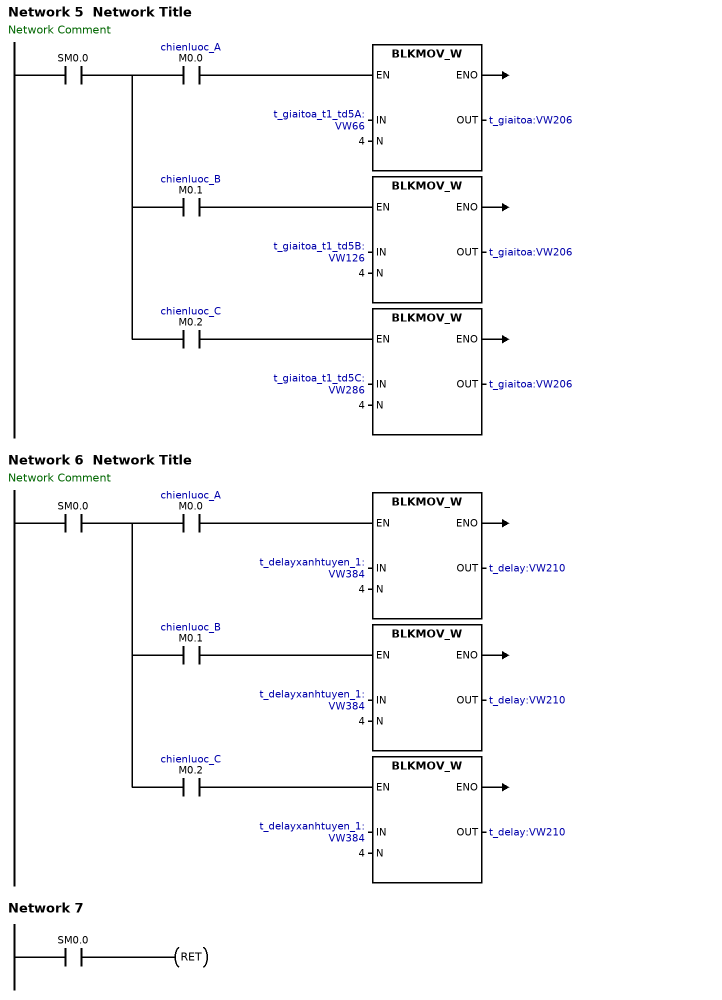
[picture p24: SBR7 networks 5-7]
Network 5 // Network Title
// Network Comment
LD     SM0.0
LPS
A      chienluoc_A:M0.0
BMW    t_giaitoa_t1_td5A:VW66, t_giaitoa:VW206, 4
LRD
A      chienluoc_B:M0.1
BMW    t_giaitoa_t1_td5B:VW126, t_giaitoa:VW206, 4
LPP
A      chienluoc_C:M0.2
BMW    t_giaitoa_t1_td5C:VW286, t_giaitoa:VW206, 4
Network 6 // Network Title
// Network Comment
LD     SM0.0
LPS
A      chienluoc_A:M0.0
BMW    t_delayxanhtuyen_1:VW384, t_delay:VW210, 4
LRD
A      chienluoc_B:M0.1
BMW    t_delayxanhtuyen_1:VW384, t_delay:VW210, 4
LPP
A      chienluoc_C:M0.2
BMW    t_delayxanhtuyen_1:VW384, t_delay:VW210, 4
Network 7
LD     SM0.0
CRET
END_SUBROUTINE_BLOCK

SUBROUTINE_BLOCK thoidiem6:SBR8
TITLE=SUBROUTINE COMMENTS
BEGIN
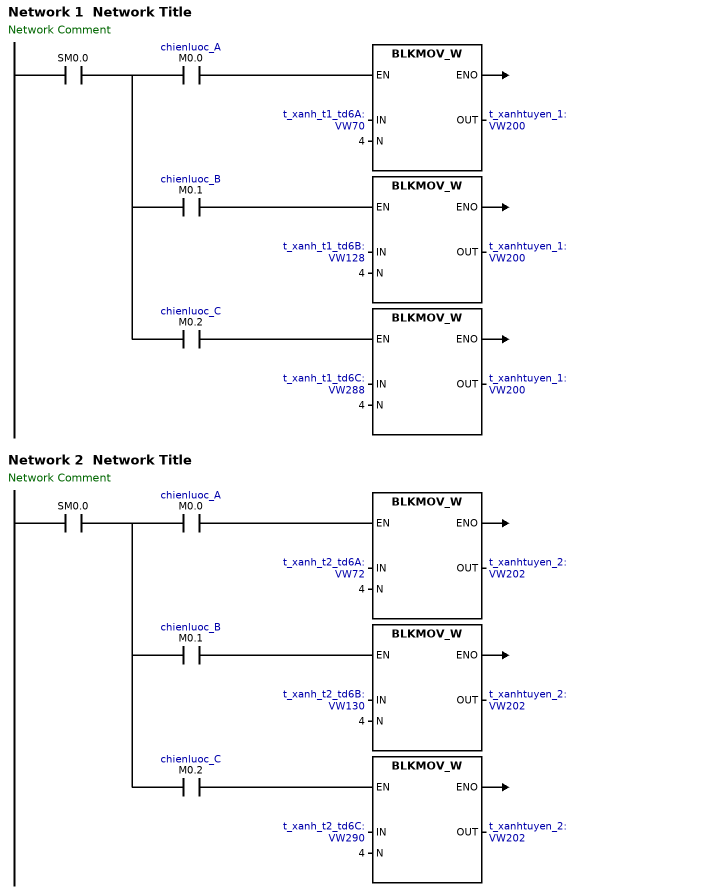
Network 1 // Network Title
// Network Comment
LD     SM0.0
LPS
A      chienluoc_A:M0.0
BMW    t_xanh_t1_td6A:VW70, t_xanhtuyen_1:VW200, 4
LRD
A      chienluoc_B:M0.1
BMW    t_xanh_t1_td6B:VW128, t_xanhtuyen_1:VW200, 4
LPP
A      chienluoc_C:M0.2
BMW    t_xanh_t1_td6C:VW288, t_xanhtuyen_1:VW200, 4
Network 2 // Network Title
// Network Comment
LD     SM0.0
LPS
A      chienluoc_A:M0.0
BMW    t_xanh_t2_td6A:VW72, t_xanhtuyen_2:VW202, 4
LRD
A      chienluoc_B:M0.1
BMW    t_xanh_t2_td6B:VW130, t_xanhtuyen_2:VW202, 4
LPP
A      chienluoc_C:M0.2
BMW    t_xanh_t2_td6C:VW290, t_xanhtuyen_2:VW202, 4
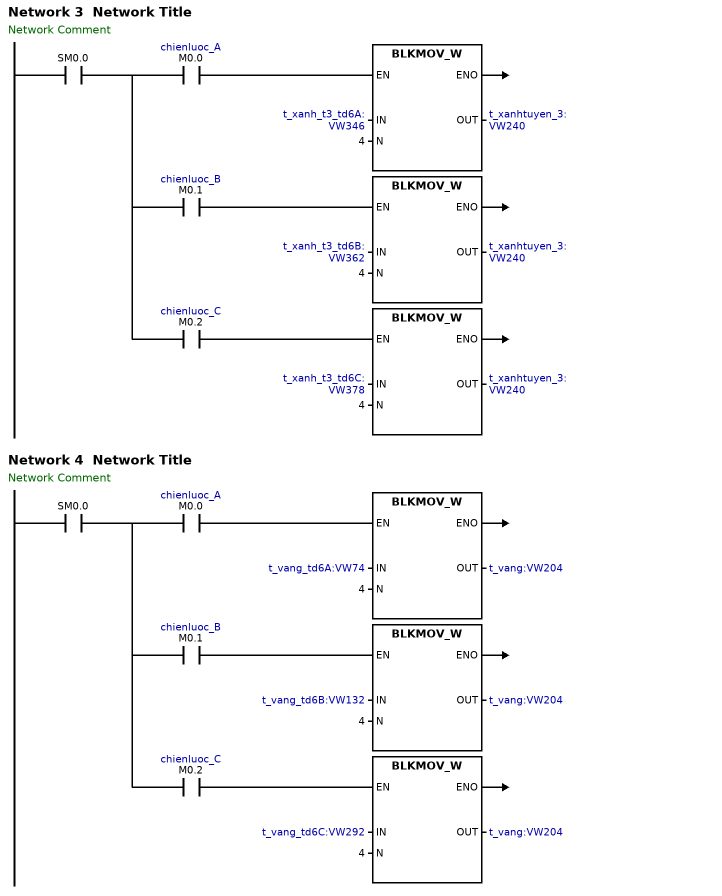
Network 3 // Network Title
// Network Comment
LD     SM0.0
LPS
A      chienluoc_A:M0.0
BMW    t_xanh_t3_td6A:VW346, t_xanhtuyen_3:VW240, 4
LRD
A      chienluoc_B:M0.1
BMW    t_xanh_t3_td6B:VW362, t_xanhtuyen_3:VW240, 4
LPP
A      chienluoc_C:M0.2
BMW    t_xanh_t3_td6C:VW378, t_xanhtuyen_3:VW240, 4
Network 4 // Network Title
// Network Comment
LD     SM0.0
LPS
A      chienluoc_A:M0.0
BMW    t_vang_td6A:VW74, t_vang:VW204, 4
LRD
A      chienluoc_B:M0.1
BMW    t_vang_td6B:VW132, t_vang:VW204, 4
LPP
A      chienluoc_C:M0.2
BMW    t_vang_td6C:VW292, t_vang:VW204, 4
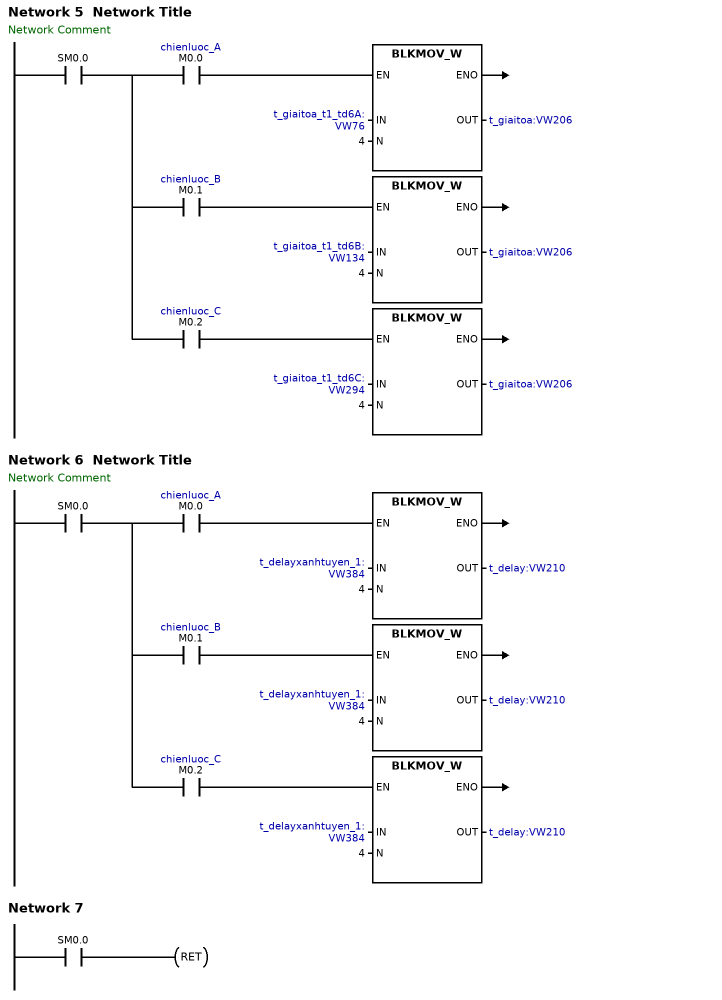
Network 5 // Network Title
// Network Comment
LD     SM0.0
LPS
A      chienluoc_A:M0.0
BMW    t_giaitoa_t1_td6A:VW76, t_giaitoa:VW206, 4
LRD
A      chienluoc_B:M0.1
BMW    t_giaitoa_t1_td6B:VW134, t_giaitoa:VW206, 4
LPP
A      chienluoc_C:M0.2
BMW    t_giaitoa_t1_td6C:VW294, t_giaitoa:VW206, 4
Network 6 // Network Title
// Network Comment
LD     SM0.0
LPS
A      chienluoc_A:M0.0
BMW    t_delayxanhtuyen_1:VW384, t_delay:VW210, 4
LRD
A      chienluoc_B:M0.1
BMW    t_delayxanhtuyen_1:VW384, t_delay:VW210, 4
LPP
A      chienluoc_C:M0.2
BMW    t_delayxanhtuyen_1:VW384, t_delay:VW210, 4
Network 7
LD     SM0.0
CRET
END_SUBROUTINE_BLOCK

SUBROUTINE_BLOCK thoidiem7:SBR9
TITLE=SUBROUTINE COMMENTS
BEGIN
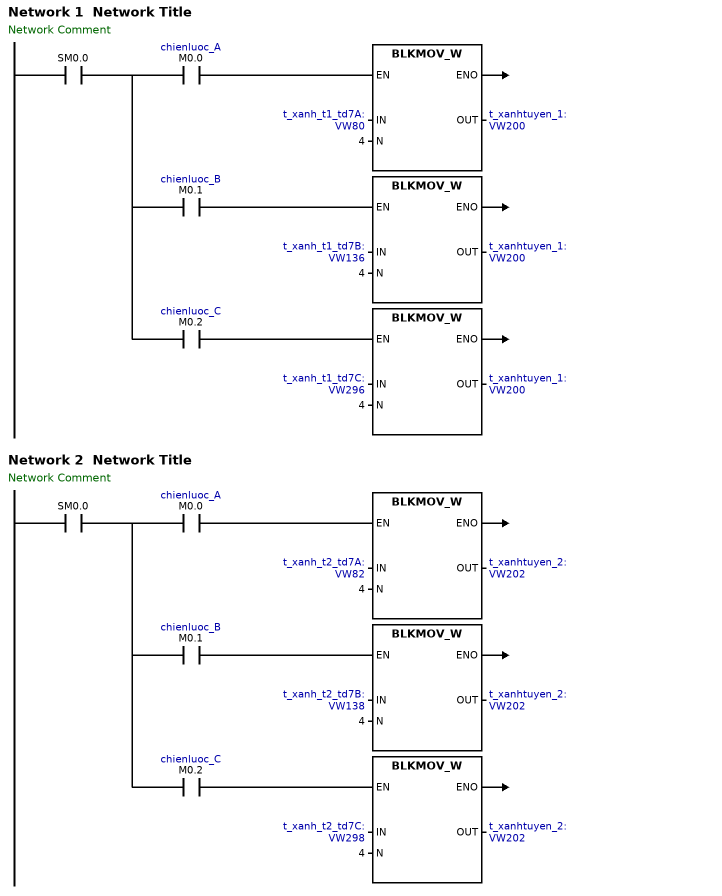
Network 1 // Network Title
// Network Comment
LD     SM0.0
LPS
A      chienluoc_A:M0.0
BMW    t_xanh_t1_td7A:VW80, t_xanhtuyen_1:VW200, 4
LRD
A      chienluoc_B:M0.1
BMW    t_xanh_t1_td7B:VW136, t_xanhtuyen_1:VW200, 4
LPP
A      chienluoc_C:M0.2
BMW    t_xanh_t1_td7C:VW296, t_xanhtuyen_1:VW200, 4
Network 2 // Network Title
// Network Comment
LD     SM0.0
LPS
A      chienluoc_A:M0.0
BMW    t_xanh_t2_td7A:VW82, t_xanhtuyen_2:VW202, 4
LRD
A      chienluoc_B:M0.1
BMW    t_xanh_t2_td7B:VW138, t_xanhtuyen_2:VW202, 4
LPP
A      chienluoc_C:M0.2
BMW    t_xanh_t2_td7C:VW298, t_xanhtuyen_2:VW202, 4
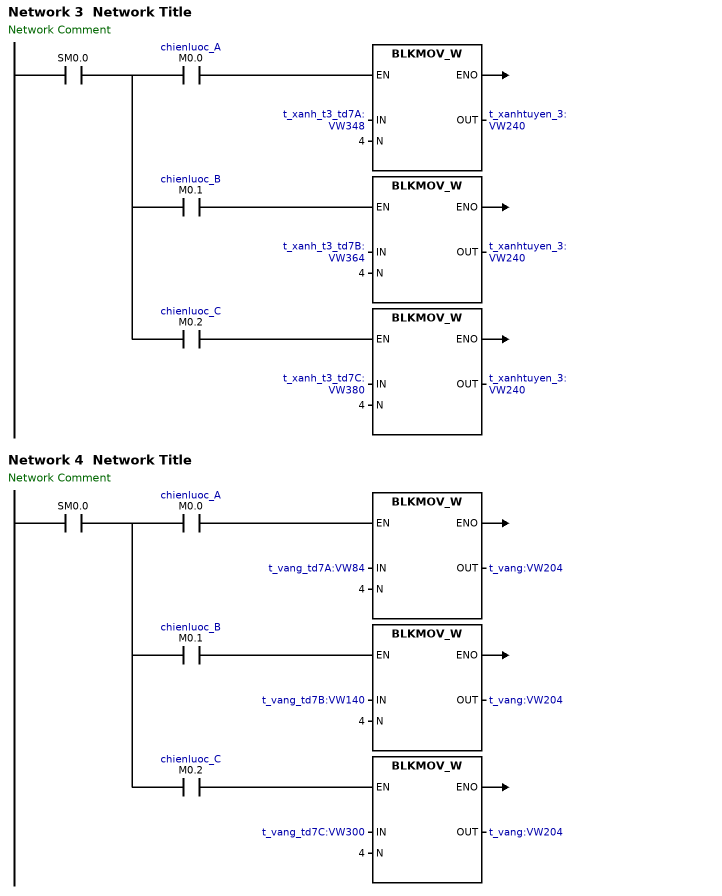
Network 3 // Network Title
// Network Comment
LD     SM0.0
LPS
A      chienluoc_A:M0.0
BMW    t_xanh_t3_td7A:VW348, t_xanhtuyen_3:VW240, 4
LRD
A      chienluoc_B:M0.1
BMW    t_xanh_t3_td7B:VW364, t_xanhtuyen_3:VW240, 4
LPP
A      chienluoc_C:M0.2
BMW    t_xanh_t3_td7C:VW380, t_xanhtuyen_3:VW240, 4
Network 4 // Network Title
// Network Comment
LD     SM0.0
LPS
A      chienluoc_A:M0.0
BMW    t_vang_td7A:VW84, t_vang:VW204, 4
LRD
A      chienluoc_B:M0.1
BMW    t_vang_td7B:VW140, t_vang:VW204, 4
LPP
A      chienluoc_C:M0.2
BMW    t_vang_td7C:VW300, t_vang:VW204, 4
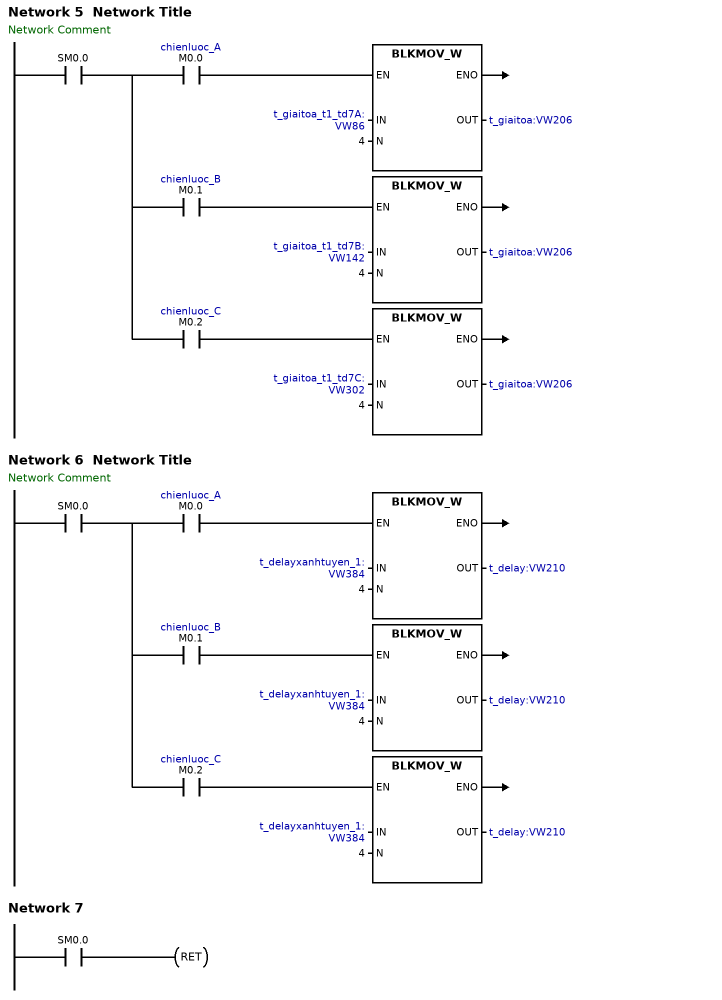
Network 5 // Network Title
// Network Comment
LD     SM0.0
LPS
A      chienluoc_A:M0.0
BMW    t_giaitoa_t1_td7A:VW86, t_giaitoa:VW206, 4
LRD
A      chienluoc_B:M0.1
BMW    t_giaitoa_t1_td7B:VW142, t_giaitoa:VW206, 4
LPP
A      chienluoc_C:M0.2
BMW    t_giaitoa_t1_td7C:VW302, t_giaitoa:VW206, 4
Network 6 // Network Title
// Network Comment
LD     SM0.0
LPS
A      chienluoc_A:M0.0
BMW    t_delayxanhtuyen_1:VW384, t_delay:VW210, 4
LRD
A      chienluoc_B:M0.1
BMW    t_delayxanhtuyen_1:VW384, t_delay:VW210, 4
LPP
A      chienluoc_C:M0.2
BMW    t_delayxanhtuyen_1:VW384, t_delay:VW210, 4
Network 7
LD     SM0.0
CRET
END_SUBROUTINE_BLOCK

SUBROUTINE_BLOCK chonngay:SBR11
TITLE=SUBROUTINE COMMENTS
BEGIN
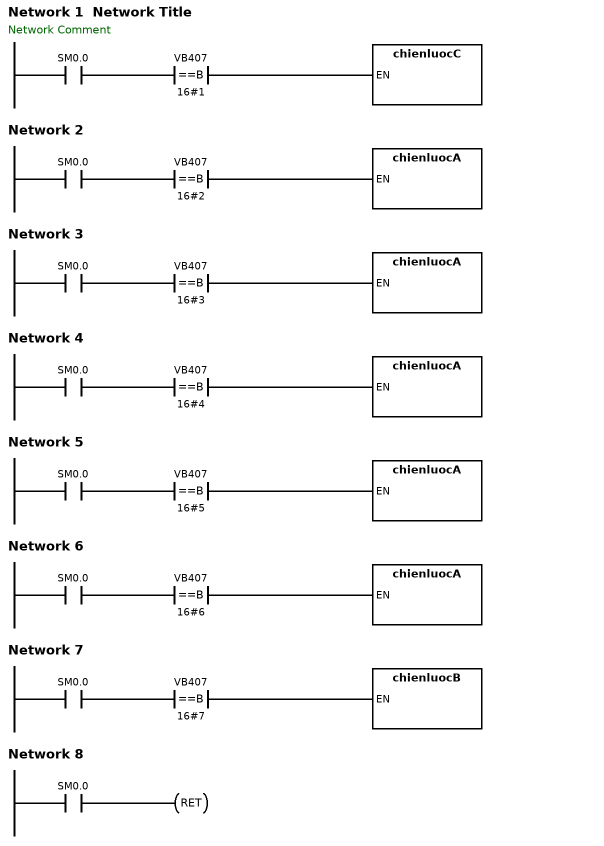
Network 1 // Network Title
// Network Comment
LD     SM0.0
AB=    VB407, 16#1
CALL   chienluocC:SBR15
Network 2
LD     SM0.0
AB=    VB407, 16#2
CALL   chienluocA:SBR12
Network 3
LD     SM0.0
AB=    VB407, 16#3
CALL   chienluocA:SBR12
Network 4
LD     SM0.0
AB=    VB407, 16#4
CALL   chienluocA:SBR12
Network 5
LD     SM0.0
AB=    VB407, 16#5
CALL   chienluocA:SBR12
Network 6
LD     SM0.0
AB=    VB407, 16#6
CALL   chienluocA:SBR12
Network 7
LD     SM0.0
AB=    VB407, 16#7
CALL   chienluocB:SBR13
Network 8
LD     SM0.0
CRET
END_SUBROUTINE_BLOCK

SUBROUTINE_BLOCK chienluocA:SBR12
TITLE=SUBROUTINE COMMENTS
BEGIN
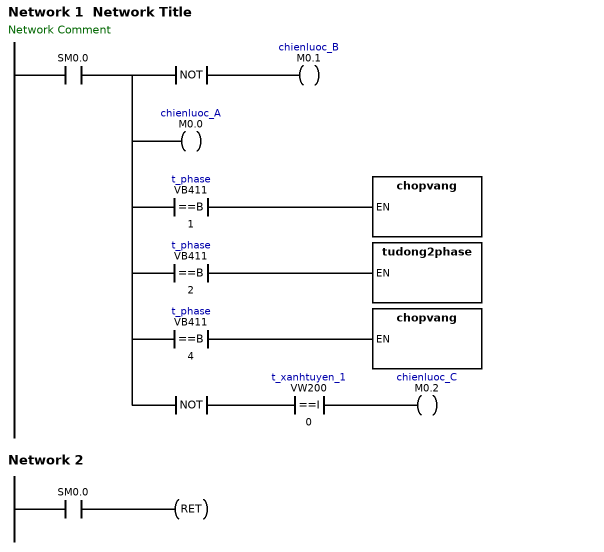
Network 1 // Network Title
// Network Comment
LD     SM0.0
LPS
NOT
=      chienluoc_B:M0.1
LRD
=      chienluoc_A:M0.0
LRD
AB=    t_phase:VB411, 1
CALL   chopvang:SBR1
LRD
AB=    t_phase:VB411, 2
CALL   tudong2phase:SBR0
LRD
AB=    t_phase:VB411, 4
CALL   chopvang:SBR1
LPP
NOT
AW=    t_xanhtuyen_1:VW200, 0
=      chienluoc_C:M0.2
Network 2
LD     SM0.0
CRET
END_SUBROUTINE_BLOCK

SUBROUTINE_BLOCK chienluocB:SBR13
TITLE=SUBROUTINE COMMENTS
BEGIN
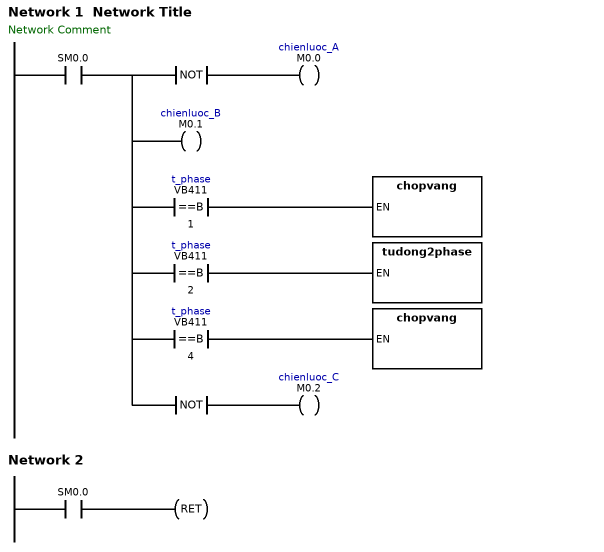
Network 1 // Network Title
// Network Comment
LD     SM0.0
LPS
NOT
=      chienluoc_A:M0.0
LRD
=      chienluoc_B:M0.1
LRD
AB=    t_phase:VB411, 1
CALL   chopvang:SBR1
LRD
AB=    t_phase:VB411, 2
CALL   tudong2phase:SBR0
LRD
AB=    t_phase:VB411, 4
CALL   chopvang:SBR1
LPP
NOT
=      chienluoc_C:M0.2
Network 2
LD     SM0.0
CRET
END_SUBROUTINE_BLOCK

SUBROUTINE_BLOCK thoidiem8:SBR14
TITLE=
BEGIN
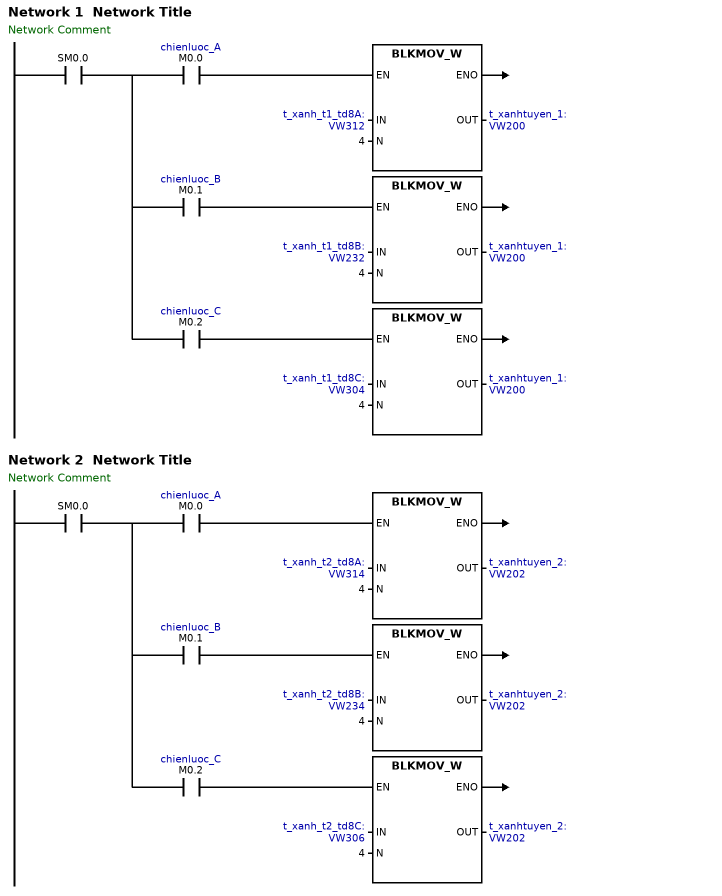
Network 1 // Network Title
// Network Comment
LD     SM0.0
LPS
A      chienluoc_A:M0.0
BMW    t_xanh_t1_td8A:VW312, t_xanhtuyen_1:VW200, 4
LRD
A      chienluoc_B:M0.1
BMW    t_xanh_t1_td8B:VW232, t_xanhtuyen_1:VW200, 4
LPP
A      chienluoc_C:M0.2
BMW    t_xanh_t1_td8C:VW304, t_xanhtuyen_1:VW200, 4
Network 2 // Network Title
// Network Comment
LD     SM0.0
LPS
A      chienluoc_A:M0.0
BMW    t_xanh_t2_td8A:VW314, t_xanhtuyen_2:VW202, 4
LRD
A      chienluoc_B:M0.1
BMW    t_xanh_t2_td8B:VW234, t_xanhtuyen_2:VW202, 4
LPP
A      chienluoc_C:M0.2
BMW    t_xanh_t2_td8C:VW306, t_xanhtuyen_2:VW202, 4
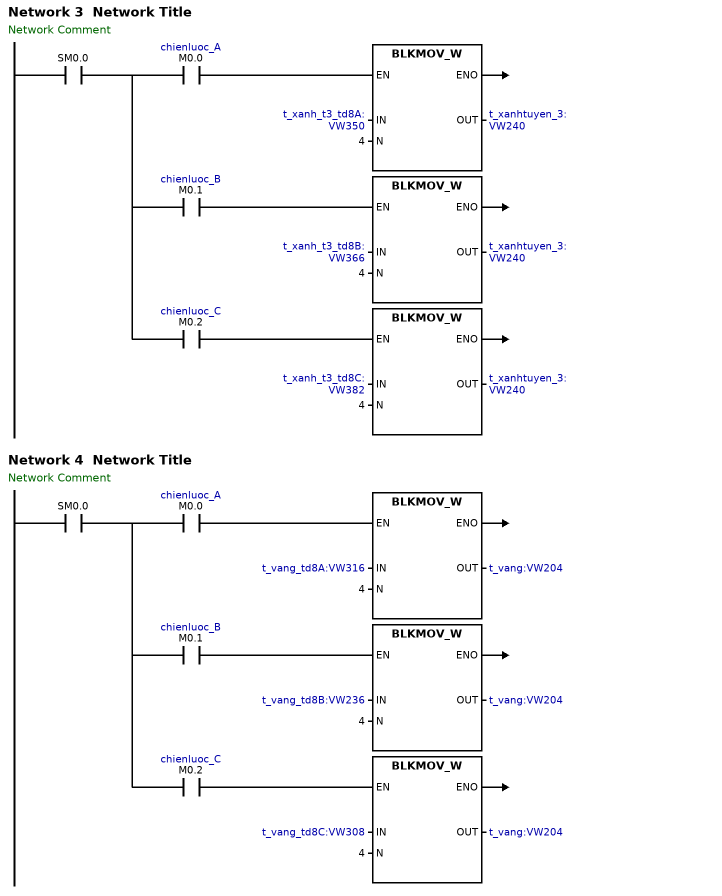
Network 3 // Network Title
// Network Comment
LD     SM0.0
LPS
A      chienluoc_A:M0.0
BMW    t_xanh_t3_td8A:VW350, t_xanhtuyen_3:VW240, 4
LRD
A      chienluoc_B:M0.1
BMW    t_xanh_t3_td8B:VW366, t_xanhtuyen_3:VW240, 4
LPP
A      chienluoc_C:M0.2
BMW    t_xanh_t3_td8C:VW382, t_xanhtuyen_3:VW240, 4
Network 4 // Network Title
// Network Comment
LD     SM0.0
LPS
A      chienluoc_A:M0.0
BMW    t_vang_td8A:VW316, t_vang:VW204, 4
LRD
A      chienluoc_B:M0.1
BMW    t_vang_td8B:VW236, t_vang:VW204, 4
LPP
A      chienluoc_C:M0.2
BMW    t_vang_td8C:VW308, t_vang:VW204, 4
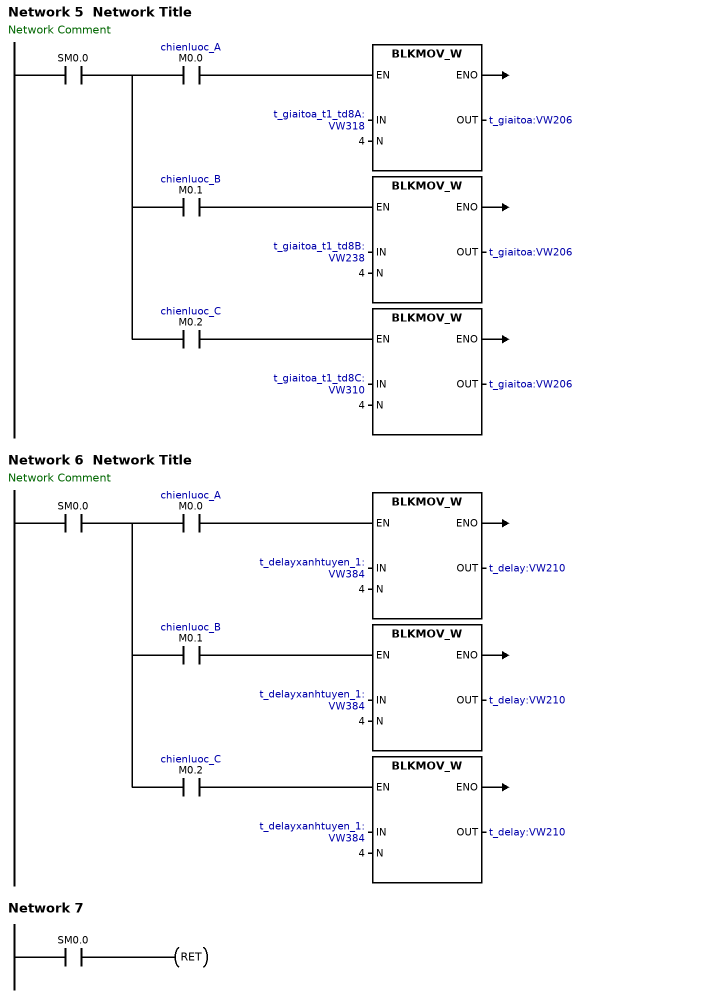
Network 5 // Network Title
// Network Comment
LD     SM0.0
LPS
A      chienluoc_A:M0.0
BMW    t_giaitoa_t1_td8A:VW318, t_giaitoa:VW206, 4
LRD
A      chienluoc_B:M0.1
BMW    t_giaitoa_t1_td8B:VW238, t_giaitoa:VW206, 4
LPP
A      chienluoc_C:M0.2
BMW    t_giaitoa_t1_td8C:VW310, t_giaitoa:VW206, 4
Network 6 // Network Title
// Network Comment
LD     SM0.0
LPS
A      chienluoc_A:M0.0
BMW    t_delayxanhtuyen_1:VW384, t_delay:VW210, 4
LRD
A      chienluoc_B:M0.1
BMW    t_delayxanhtuyen_1:VW384, t_delay:VW210, 4
LPP
A      chienluoc_C:M0.2
BMW    t_delayxanhtuyen_1:VW384, t_delay:VW210, 4
Network 7
LD     SM0.0
CRET
END_SUBROUTINE_BLOCK

SUBROUTINE_BLOCK chienluocC:SBR15
TITLE=
BEGIN
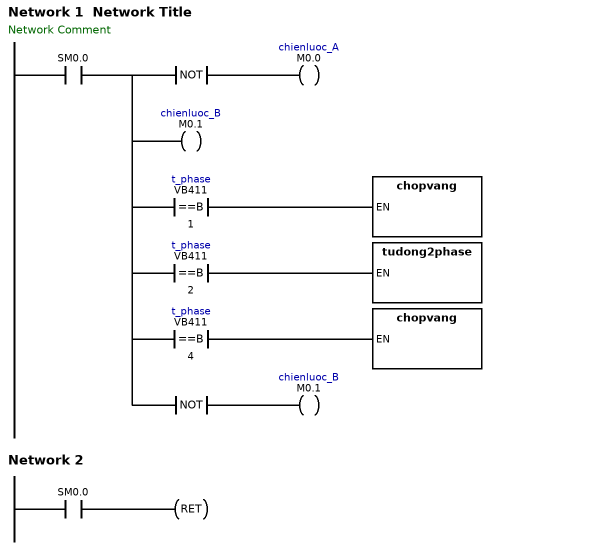
Network 1 // Network Title
// Network Comment
LD     SM0.0
LPS
NOT
=      chienluoc_A:M0.0
LRD
=      chienluoc_B:M0.1
LRD
AB=    t_phase:VB411, 1
CALL   chopvang:SBR1
LRD
AB=    t_phase:VB411, 2
CALL   tudong2phase:SBR0
LRD
AB=    t_phase:VB411, 4
CALL   chopvang:SBR1
LPP
NOT
=      chienluoc_B:M0.1
Network 2
LD     SM0.0
CRET
END_SUBROUTINE_BLOCK

SUBROUTINE_BLOCK tinhtime:SBR16
TITLE=SUBROUTINE COMMENTS
VAR_INPUT
Y0:INT;	// LW0 
END_VAR
VAR_IN_OUT
Y1:INT;	// LW2 
Y2:INT;	// LW4 
Y3:INT;	// LW6 
Y4:INT;	// LW8 
Y5:INT;	// LW10 
Y6:INT;	// LW12 
Y7:INT;	// LW14 
Y8:INT;	// LW16 
Y9:INT;	// LW18 
Y10:INT;	// LW20 
END_VAR
BEGIN
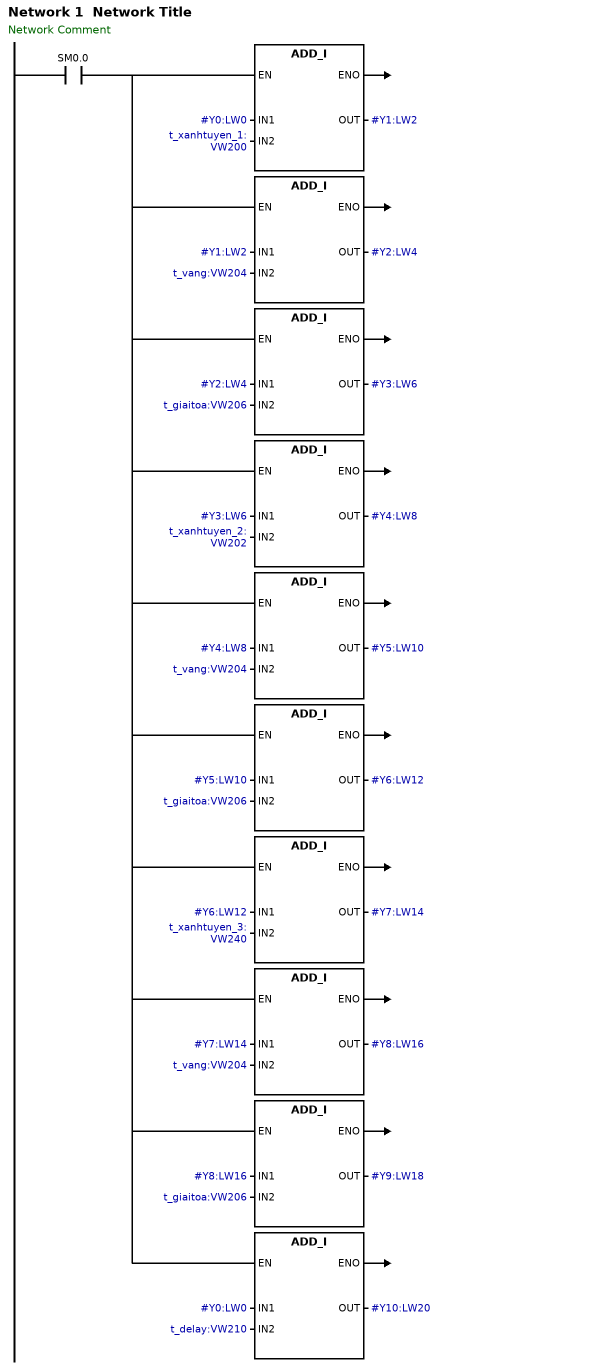
Network 1 // Network Title
// Network Comment
LD     SM0.0
MOVW   #Y0:LW0, #Y1:LW2
+I     t_xanhtuyen_1:VW200, #Y1:LW2
MOVW   #Y1:LW2, #Y2:LW4
+I     t_vang:VW204, #Y2:LW4
MOVW   #Y2:LW4, #Y3:LW6
+I     t_giaitoa:VW206, #Y3:LW6
MOVW   #Y3:LW6, #Y4:LW8
+I     t_xanhtuyen_2:VW202, #Y4:LW8
MOVW   #Y4:LW8, #Y5:LW10
+I     t_vang:VW204, #Y5:LW10
MOVW   #Y5:LW10, #Y6:LW12
+I     t_giaitoa:VW206, #Y6:LW12
MOVW   #Y6:LW12, #Y7:LW14
+I     t_xanhtuyen_3:VW240, #Y7:LW14
MOVW   #Y7:LW14, #Y8:LW16
+I     t_vang:VW204, #Y8:LW16
MOVW   #Y8:LW16, #Y9:LW18
+I     t_giaitoa:VW206, #Y9:LW18
MOVW   #Y0:LW0, #Y10:LW20
+I     t_delay:VW210, #Y10:LW20
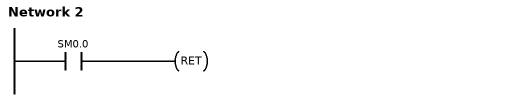
Network 2
LD     SM0.0
CRET
END_SUBROUTINE_BLOCK

SUBROUTINE_BLOCK nut_nhan_di_bo:SBR17
TITLE=SUBROUTINE COMMENTS
BEGIN
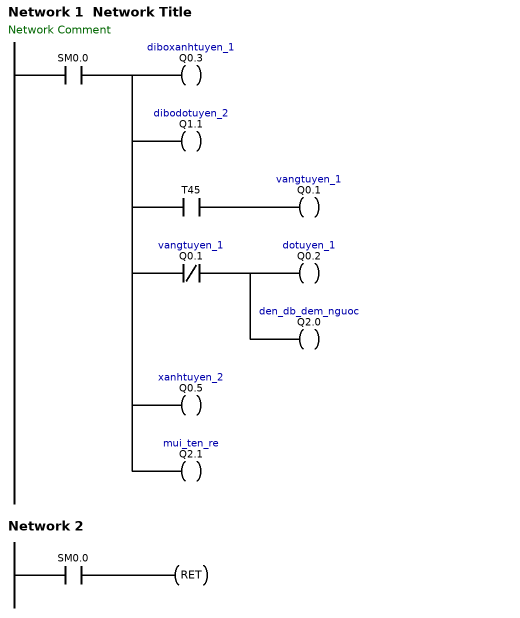
Network 1 // Network Title
// Network Comment
LD     SM0.0
LPS
=      diboxanhtuyen_1:Q0.3
=      dibodotuyen_2:Q1.1
A      T45
=      vangtuyen_1:Q0.1
LRD
AN     vangtuyen_1:Q0.1
=      dotuyen_1:Q0.2
=      den_db_dem_nguoc:Q2.0
LPP
=      xanhtuyen_2:Q0.5
=      mui_ten_re:Q2.1
Network 2
LD     SM0.0
CRET
Network 11 // Network Title
// Network Comment
END_SUBROUTINE_BLOCK

SUBROUTINE_BLOCK Set_bieumau:SBR18
TITLE=SUBROUTINE COMMENTS
BEGIN
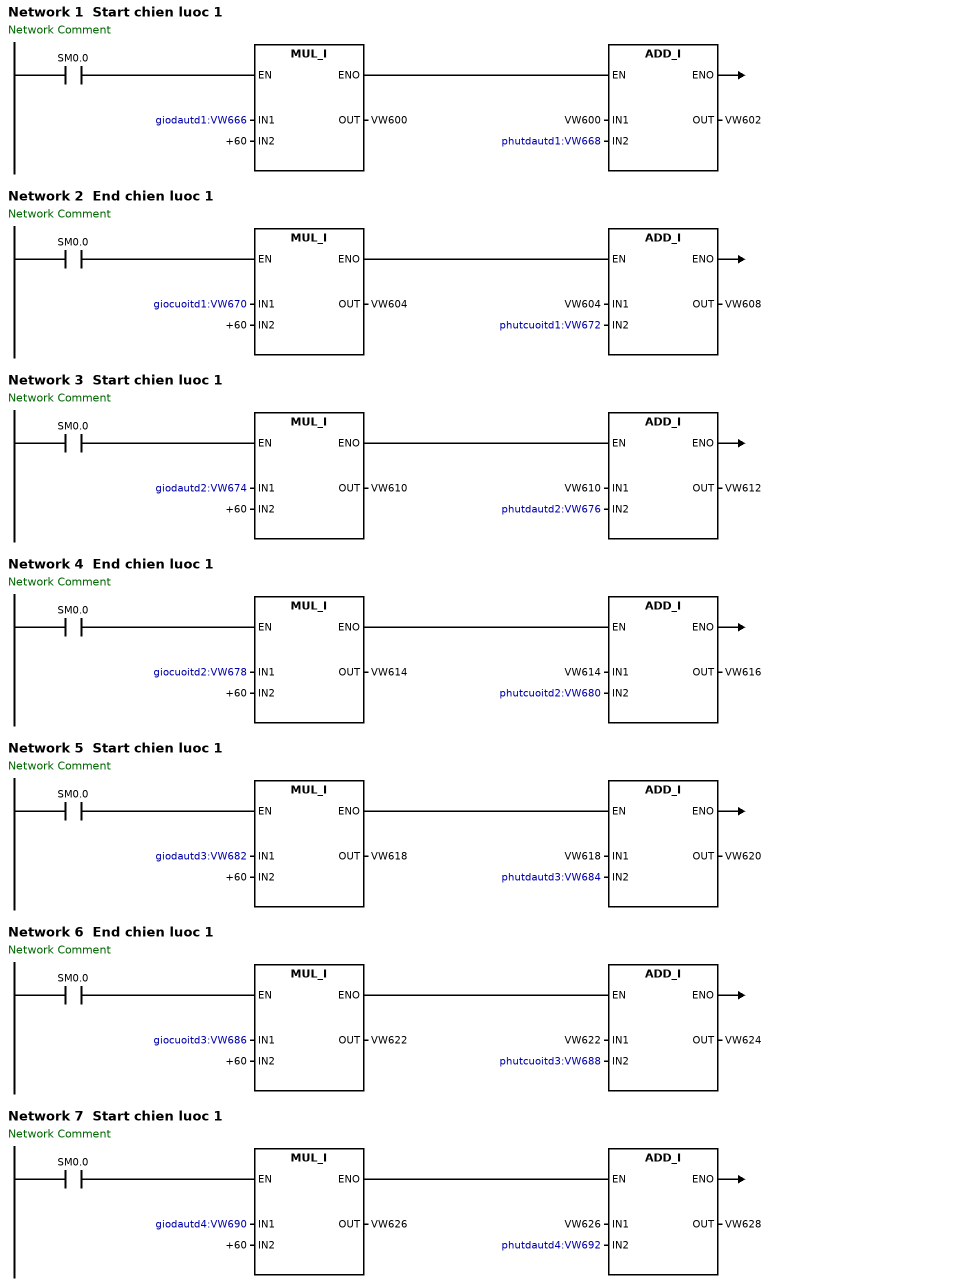
Network 1 // Start chien luoc 1
// Network Comment
LD     SM0.0
MOVW   giodautd1:VW666, VW600
AENO
*I     +60, VW600
AENO
MOVW   VW600, VW602
+I     phutdautd1:VW668, VW602
Network 2 // End chien luoc 1
// Network Comment
LD     SM0.0
MOVW   giocuoitd1:VW670, VW604
AENO
*I     +60, VW604
AENO
MOVW   VW604, VW608
+I     phutcuoitd1:VW672, VW608
Network 3 // Start chien luoc 1
// Network Comment
LD     SM0.0
MOVW   giodautd2:VW674, VW610
AENO
*I     +60, VW610
AENO
MOVW   VW610, VW612
+I     phutdautd2:VW676, VW612
Network 4 // End chien luoc 1
// Network Comment
LD     SM0.0
MOVW   giocuoitd2:VW678, VW614
AENO
*I     +60, VW614
AENO
MOVW   VW614, VW616
+I     phutcuoitd2:VW680, VW616
Network 5 // Start chien luoc 1
// Network Comment
LD     SM0.0
MOVW   giodautd3:VW682, VW618
AENO
*I     +60, VW618
AENO
MOVW   VW618, VW620
+I     phutdautd3:VW684, VW620
Network 6 // End chien luoc 1
// Network Comment
LD     SM0.0
MOVW   giocuoitd3:VW686, VW622
AENO
*I     +60, VW622
AENO
MOVW   VW622, VW624
+I     phutcuoitd3:VW688, VW624
Network 7 // Start chien luoc 1
// Network Comment
LD     SM0.0
MOVW   giodautd4:VW690, VW626
AENO
*I     +60, VW626
AENO
MOVW   VW626, VW628
+I     phutdautd4:VW692, VW628
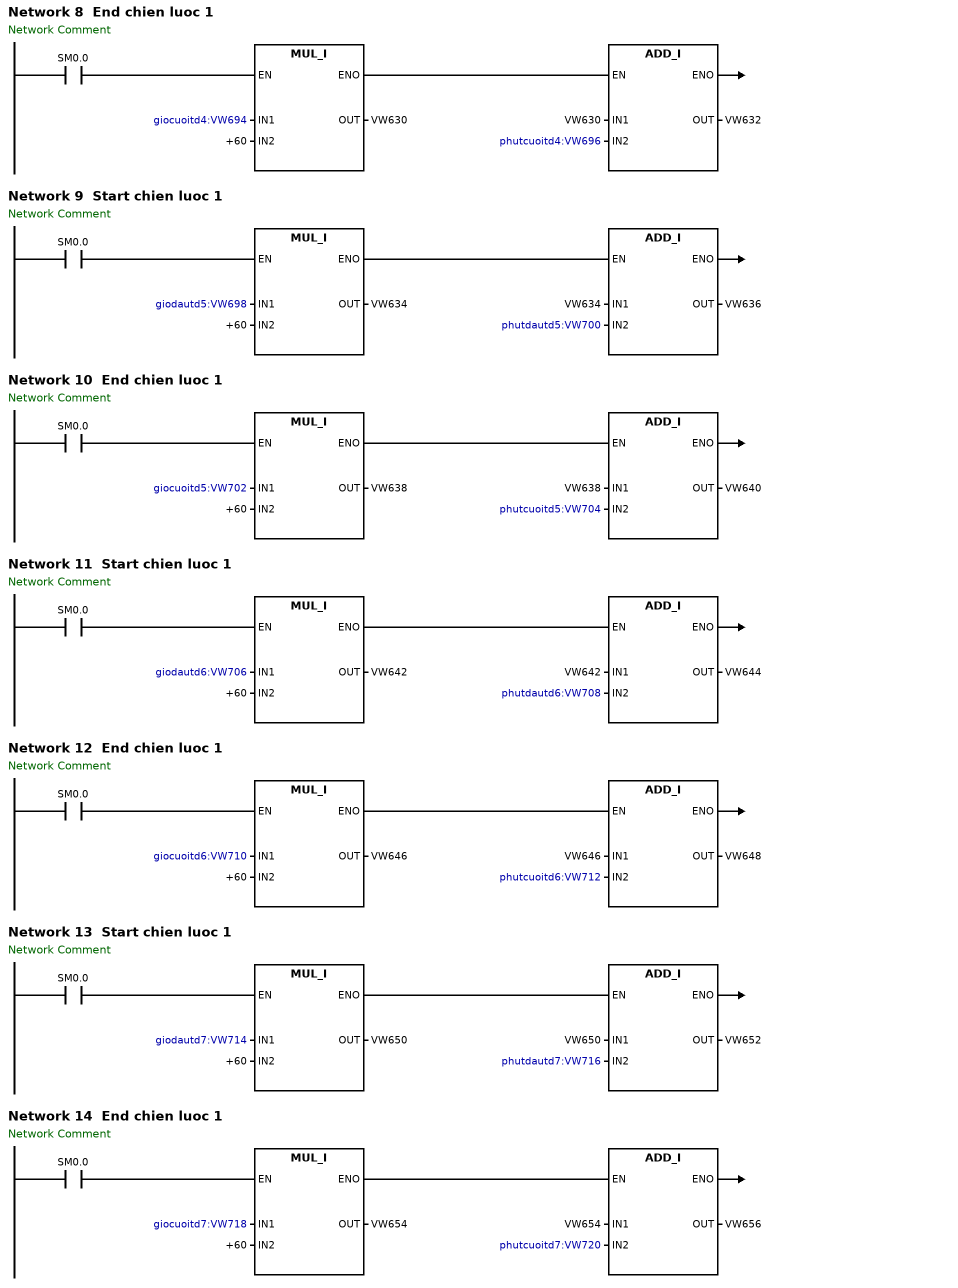
Network 8 // End chien luoc 1
// Network Comment
LD     SM0.0
MOVW   giocuoitd4:VW694, VW630
AENO
*I     +60, VW630
AENO
MOVW   VW630, VW632
+I     phutcuoitd4:VW696, VW632
Network 9 // Start chien luoc 1
// Network Comment
LD     SM0.0
MOVW   giodautd5:VW698, VW634
AENO
*I     +60, VW634
AENO
MOVW   VW634, VW636
+I     phutdautd5:VW700, VW636
Network 10 // End chien luoc 1
// Network Comment
LD     SM0.0
MOVW   giocuoitd5:VW702, VW638
AENO
*I     +60, VW638
AENO
MOVW   VW638, VW640
+I     phutcuoitd5:VW704, VW640
Network 11 // Start chien luoc 1
// Network Comment
LD     SM0.0
MOVW   giodautd6:VW706, VW642
AENO
*I     +60, VW642
AENO
MOVW   VW642, VW644
+I     phutdautd6:VW708, VW644
Network 12 // End chien luoc 1
// Network Comment
LD     SM0.0
MOVW   giocuoitd6:VW710, VW646
AENO
*I     +60, VW646
AENO
MOVW   VW646, VW648
+I     phutcuoitd6:VW712, VW648
Network 13 // Start chien luoc 1
// Network Comment
LD     SM0.0
MOVW   giodautd7:VW714, VW650
AENO
*I     +60, VW650
AENO
MOVW   VW650, VW652
+I     phutdautd7:VW716, VW652
Network 14 // End chien luoc 1
// Network Comment
LD     SM0.0
MOVW   giocuoitd7:VW718, VW654
AENO
*I     +60, VW654
AENO
MOVW   VW654, VW656
+I     phutcuoitd7:VW720, VW656
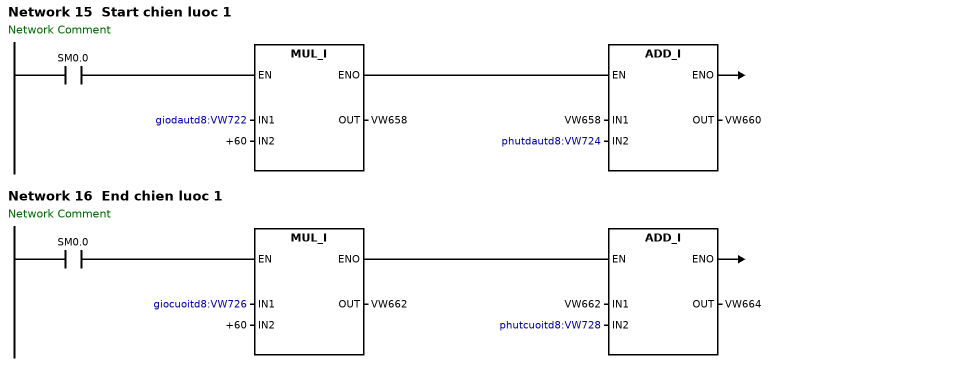
Network 15 // Start chien luoc 1
// Network Comment
LD     SM0.0
MOVW   giodautd8:VW722, VW658
AENO
*I     +60, VW658
AENO
MOVW   VW658, VW660
+I     phutdautd8:VW724, VW660
Network 16 // End chien luoc 1
// Network Comment
LD     SM0.0
MOVW   giocuoitd8:VW726, VW662
AENO
*I     +60, VW662
AENO
MOVW   VW662, VW664
+I     phutcuoitd8:VW728, VW664
END_SUBROUTINE_BLOCK

DATA_BLOCK_TAB USER1
BEGIN
//DATA PAGE COMMENTS
//Press F1 for help and example data page
//Gio he thong,nhap gio tu 16#05-16#23
         gio_on_he_thong, 16#5
         phut_on_he_thong, 16#0
         gio_off_he_thong, 16#23
         phut_off_he_thong, 16#0
         set_time, 16#0
         set_time_2, 16#0
         t_phase, 16#2
         t_dependent, 16#0
         t_delayxanhtuyen_1, +50
// LUU Y LA PHAI NHAP TAT CA CAC SO , NHO LA PHAI CO DAU + DUNG TRUOC//
//thoi gian xanh - vang - do cho thoi diem thu 1A  (tu thoi gian 05h-07h30)
         giodautd1, +5
         phutdautd1, +0
         giocuoitd1, +7
         phutcuoitd1, +0
         t_xanh_t1_td1A, +0  // gia tri thoi gian xanh tuyen 1
         t_xanh_t2_td1A, +0  // gia tri thoi gian xanh tuyen 2
         t_xanh_t3_td1A, +0  // gia tri thoi gian xanh tuyen 3
         t_vang_td1A, +50    // gia tri thoi gian vang
         t_giaitoa_t1_td1A, +0 // gia tri thoi gian giai toa
//thoi gian xanh - vang - do cho thoi diem thu 2A  (tu thoi gian 07h30-8h30)
         giodautd2, +7
         phutdautd2, +30
         giocuoitd2, +8
         phutcuoitd2, +30
         t_xanh_t1_td2A, +300 // gia tri thoi gian xanh tuyen 1
         t_xanh_t2_td2A, +200 // gia tri thoi gian xanh tuyen 2
         t_xanh_t3_td2A, +0  // gia tri thoi gian xanh tuyen 3
         t_vang_td2A, +30    // gia tri thoi gian vang
         t_giaitoa_t1_td2A, +0 // gia tri thoi gian giai toa
//thoi gian xanh - vang - do cho thoi diem thu 3A  (tu thoi gian 8h30-15h)
         giodautd3, +8
         phutdautd3, +30
         giocuoitd3, +15
         phutcuoitd3, +0
         t_xanh_t1_td3A, +0  // gia tri thoi gian xanh tuyen 1
         t_xanh_t2_td3A, +0  // gia tri thoi gian xanh tuyen 2
         t_xanh_t3_td3A, +0  // gia tri thoi gian xanh tuyen 3
         t_vang_td3A, +50    // gia tri thoi gian vang
         t_giaitoa_t1_td3A, +0 // gia tri thoi gian giai toa
//thoi gian xanh - vang - do cho thoi diem thu 4A  (tu thoi gian 15h0-16h30)
         giodautd4, +15
         phutdautd4, +0
         giocuoitd4, +16
         phutcuoitd4, +30
         t_xanh_t1_td4A, +300 // gia tri thoi gian xanh tuyen 1
         t_xanh_t2_td4A, +200 // gia tri thoi gian xanh tuyen 2
         t_xanh_t3_td4A, +0  // gia tri thoi gian xanh tuyen 3
         t_vang_td4A, +30    // gia tri thoi gian vang
         t_giaitoa_t1_td4A, +0 // gia tri thoi gian giai toa
//thoi gian xanh - vang - do cho thoi diem thu 5A  (tu thoi gian 16h30-19h)
         giodautd5, +16
         phutdautd5, +30
         giocuoitd5, +19
         phutcuoitd5, +0
         t_xanh_t1_td5A, +0  // gia tri thoi gian xanh tuyen 1
         t_xanh_t2_td5A, +0  // gia tri thoi gian xanh tuyen 2
         t_xanh_t3_td5A, +0  // gia tri thoi gian xanh tuyen 3
         t_vang_td5A, +50    // gia tri thoi gian vang
         t_giaitoa_t1_td5A, +0 // gia tri thoi gian giai toa
//thoi gian xanh - vang - do cho thoi diem thu 6A  (tu thoi gian 19h-20h)
         giodautd6, +19
         phutdautd6, +0
         giocuoitd6, +20
         phutcuoitd6, +0
         t_xanh_t1_td6A, +0  // gia tri thoi gian xanh tuyen 1
         t_xanh_t2_td6A, +0  // gia tri thoi gian xanh tuyen 2
         t_xanh_t3_td6A, +0  // gia tri thoi gian xanh tuyen 3
         t_vang_td6A, +50    // gia tri thoi gian vang
         t_giaitoa_t1_td6A, +0 // gia tri thoi gian giai toa
//thoi gian xanh - vang - do cho thoi diem thu 7A  (tu thoi gian 20h-21h)
         giodautd7, +20
         phutdautd7, +0
         giocuoitd7, +21
         phutcuoitd7, +0
         t_xanh_t1_td7A, +0  // gia tri thoi gian xanh tuyen 1
         t_xanh_t2_td7A, +0  // gia tri thoi gian xanh tuyen 2
         t_xanh_t3_td7A, +0  // gia tri thoi gian xanh tuyen 3
         t_vang_td7A, +50    // gia tri thoi gian vang
         t_giaitoa_t1_td7A, +0 // gia tri thoi gian giai toa
//thoi gian xanh - vang - do cho thoi diem thu 8A  (tu thoi gian 21h-22h)
         giodautd8, +21
         phutdautd8, +0
         giocuoitd8, +22
         phutcuoitd8, +0
         t_xanh_t1_td8A, +0  // gia tri thoi gian xanh tuyen 1
         t_xanh_t2_td8A, +0  // gia tri thoi gian xanh tuyen 2
         t_xanh_t3_td8A, +0  // gia tri thoi gian xanh tuyen 3
         t_vang_td8A, +50    // gia tri thoi gian vang
         t_giaitoa_t1_td8A, +0 // gia tri thoi gian giai toa
//*******************************************************************
//thoi gian xanh - vang - do cho thoi diem thu 1 B (tu thoi gian 06h-7h30)
         t_xanh_t1_td1B, +0  // gia tri thoi gian xanh tuyen 1
         t_xanh_t2_td1B, +0  // gia tri thoi gian xanh tuyen 2
         t_xanh_t3_td1B, +0  // gia tri thoi gian xanh tuyen 3
         t_vang_td1B, +50    // gia tri thoi gian vang
         t_giaitoa_t1_td1B, +0 // gia tri thoi gian giai toa
//thoi gian xanh - vang - do cho thoi diem thu 2 B (tu thoi gian 7h30-8h30)
         t_xanh_t1_td2B, +300 // gia tri thoi gian xanh tuyen 1
         t_xanh_t2_td2B, +200 // gia tri thoi gian xanh tuyen 2
         t_xanh_t3_td2B, +0  // gia tri thoi gian xanh tuyen 3
         t_vang_td2B, +30    // gia tri thoi gian vang
         t_giaitoa_t1_td2B, +0 // gia tri thoi gian giai toa
//thoi gian xanh - vang - do cho thoi diem thu 3 B (tu thoi gian 8h30-13h)
         t_xanh_t1_td3B, +0  // gia tri thoi gian xanh tuyen 1
         t_xanh_t2_td3B, +0  // gia tri thoi gian xanh tuyen 2
         t_xanh_t3_td3B, +0  // gia tri thoi gian xanh tuyen 3
         t_vang_td3B, +50    // gia tri thoi gian vang
         t_giaitoa_t1_td3B, +0 // gia tri thoi gian giai toa
//thoi gian xanh - vang - do cho thoi diem thu 4 B (tu thoi gian 13h-15h)
         t_xanh_t1_td4B, +0  // gia tri thoi gian xanh tuyen 1
         t_xanh_t2_td4B, +0  // gia tri thoi gian xanh tuyen 2
         t_xanh_t3_td4B, +0  // gia tri thoi gian xanh tuyen 3
         t_vang_td4B, +50    // gia tri thoi gian vang
         t_giaitoa_t1_td4B, +0 // gia tri thoi gian giai toa
//thoi gian xanh - vang - do cho thoi diem thu 5 B (tu thoi gian 15h-16h30)
         t_xanh_t1_td5B, +300 // gia tri thoi gian xanh tuyen 1
         t_xanh_t2_td5B, +200 // gia tri thoi gian xanh tuyen 2
         t_xanh_t3_td5B, +0  // gia tri thoi gian xanh tuyen 3
         t_vang_td5B, +30    // gia tri thoi gian vang
         t_giaitoa_t1_td5B, +0 // gia tri thoi gian giai toa
//thoi gian xanh - vang - do cho thoi diem thu 6 B (tu thoi gian 16h30-20h)
         t_xanh_t1_td6B, +0  // gia tri thoi gian xanh tuyen 1
         t_xanh_t2_td6B, +0  // gia tri thoi gian xanh tuyen 2
         t_xanh_t3_td6B, +0  // gia tri thoi gian xanh tuyen 3
         t_vang_td6B, +50    // gia tri thoi gian vang
         t_giaitoa_t1_td6B, +0 // gia tri thoi gian giai toa
//thoi gian xanh - vang - do cho thoi diem thu 7 B (tu thoi gian 20h-21h)
         t_xanh_t1_td7B, +0  // gia tri thoi gian xanh tuyen 1
         t_xanh_t2_td7B, +0  // gia tri thoi gian xanh tuyen 2
         t_xanh_t3_td7B, +0  // gia tri thoi gian xanh tuyen 3
         t_vang_td7B, +50    // gia tri thoi gian vang
         t_giaitoa_t1_td7B, +0 // gia tri thoi gian giai toa
//thoi gian xanh - vang - do cho thoi diem thu 8 B (tu thoi gian 21h-22h)
         t_xanh_t1_td8B, +0  // gia tri thoi gian xanh tuyen 1
         t_xanh_t2_td8B, +0  // gia tri thoi gian xanh tuyen 2
         t_xanh_t3_td8B, +0  // gia tri thoi gian xanh tuyen 3
         t_vang_td8B, +50    // gia tri thoi gian vang
         t_giaitoa_t1_td8B, +0 // gia tri thoi gian giai toa
//*******************************************************************
//thoi gian xanh - vang - do cho thoi diem thu 1 C (tu thoi gian 06h-7h30)
         t_xanh_t1_td1C, +0  // gia tri thoi gian xanh tuyen 1
         t_xanh_t2_td1C, +0  // gia tri thoi gian xanh tuyen 2
         t_xanh_t3_td1C, +0  // gia tri thoi gian xanh tuyen 3
         t_vang_td1C, +50    // gia tri thoi gian vang
         t_giaitoa_t1_td1C, +0 // gia tri thoi gian giai toa
//thoi gian xanh - vang - do cho thoi diem thu 2 C (tu thoi gian 7h30-8h30)
         t_xanh_t1_td2C, +300 // gia tri thoi gian xanh tuyen 1
         t_xanh_t2_td2C, +200 // gia tri thoi gian xanh tuyen 2
         t_xanh_t3_td2C, +0  // gia tri thoi gian xanh tuyen 3
         t_vang_td2C, +30    // gia tri thoi gian vang
         t_giaitoa_t1_td2C, +0 // gia tri thoi gian giai toa
//thoi gian xanh - vang - do cho thoi diem thu 3 C (tu thoi gian 8h30-13h)
         t_xanh_t1_td3C, +0  // gia tri thoi gian xanh tuyen 1
         t_xanh_t2_td3C, +0  // gia tri thoi gian xanh tuyen 2
         t_xanh_t3_td3C, +0  // gia tri thoi gian xanh tuyen 3
         t_vang_td3C, +50    // gia tri thoi gian vang
         t_giaitoa_t1_td3C, +0 // gia tri thoi gian giai toa
//thoi gian xanh - vang - do cho thoi diem thu 4 C (tu thoi gian 13h-15h)
         t_xanh_t1_td4C, +0  // gia tri thoi gian xanh tuyen 1
         t_xanh_t2_td4C, +0  // gia tri thoi gian xanh tuyen 2
         t_xanh_t3_td4C, +0  // gia tri thoi gian xanh tuyen 3
         t_vang_td4C, +50    // gia tri thoi gian vang
         t_giaitoa_t1_td4C, +0 // gia tri thoi gian giai toa
//thoi gian xanh - vang - do cho thoi diem thu 5 C (tu thoi gian 15h-16h30)
         t_xanh_t1_td5C, +300 // gia tri thoi gian xanh tuyen 1
         t_xanh_t2_td5C, +200 // gia tri thoi gian xanh tuyen 2
         t_xanh_t3_td5C, +0  // gia tri thoi gian xanh tuyen 3
         t_vang_td5C, +30    // gia tri thoi gian vang
         t_giaitoa_t1_td5C, +0 // gia tri thoi gian giai toa
//thoi gian xanh - vang - do cho thoi diem thu 6 C (tu thoi gian 16h30-20h)
         t_xanh_t1_td6C, +0  // gia tri thoi gian xanh tuyen 1
         t_xanh_t2_td6C, +0  // gia tri thoi gian xanh tuyen 2
         t_xanh_t3_td6C, +0  // gia tri thoi gian xanh tuyen 3
         t_vang_td6C, +50    // gia tri thoi gian vang
         t_giaitoa_t1_td6C, +0 // gia tri thoi gian giai toa
//thoi gian xanh - vang - do cho thoi diem thu 7 C (tu thoi gian 20h-21h)
         t_xanh_t1_td7C, +0  // gia tri thoi gian xanh tuyen 1
         t_xanh_t2_td7C, +0  // gia tri thoi gian xanh tuyen 2
         t_xanh_t3_td7C, +0  // gia tri thoi gian xanh tuyen 3
         t_vang_td7C, +50    // gia tri thoi gian vang
         t_giaitoa_t1_td7C, +0 // gia tri thoi gian giai toa
//thoi gian xanh - vang - do cho thoi diem thu 8 C (tu thoi gian 21h-22h)
         t_xanh_t1_td8C, +0  // gia tri thoi gian xanh tuyen 1
         t_xanh_t2_td8C, +0  // gia tri thoi gian xanh tuyen 2
         t_xanh_t3_td8C, +0  // gia tri thoi gian xanh tuyen 3
         t_vang_td8C, +50    // gia tri thoi gian vang
         t_giaitoa_t1_td8C, +0 // gia tri thoi gian giai toa
// thoi gian dem nguoc nut nhan di bo
         t_walking, +330     // gia tri thoi gian dem nguoc di bo 300 và phai cong them 30 cua thoi gian vang 
         t_vang_walking, +30 // gia tri thoi gian vang dem nguoc sau khi nhan nut di bo
//////////////////fake data
         t_setup_to_start, +100 // chop vang truoc khi start
END_DATA_BLOCK_TAB
